# EPICS autosave request: BPMApp/Db/BPMPos_settings.req
$(P)$(R)$(ACQ)$(ARRAY_NAME_CAL)ArrayCoeff-SP
